Staubli VAL3: EnterPageKey.pgx

program EnterPageKey(num& x_nKey, num& x_nSelect, string& x_sItem)
  local string l_sStr
  local num l_nKey
  local string l_sEmpty
  local string l_sValue
  local num l_nItem
  local num l_nView
  local string l_sItem
  local point lp
  local string l_sYN[2]
  local bool l_bRes
begin
  //
  switch x_nSelect
    case 0
      if x_nKey==270
        call user:editNum(x_sItem,sListItemValue[x_nSelect],fFrame[sItem].trsf.x,x_nSelect)
      endIf
    break
    case 1
      if x_nKey==270
        call user:editNum(x_sItem,sListItemValue[x_nSelect],fFrame[sItem].trsf.y,x_nSelect)
      endIf
    break
    case 2
      if x_nKey==270
         call user:editNum(x_sItem,sListItemValue[x_nSelect],fFrame[sItem].trsf.z,x_nSelect)
      endIf
    break
    case 3
      if x_nKey==270
        call user:editNum(x_sItem,sListItemValue[x_nSelect],fFrame[sItem].trsf.rx,x_nSelect)
      endIf
    break
    case 4
      if x_nKey==27
         call user:editNum(x_sItem,sListItemValue[x_nSelect],fFrame[sItem].trsf.ry,x_nSelect)
      endIf
    break
    case 5
      if x_nKey==270
        call user:editNum(x_sItem,sListItemValue[x_nSelect],fFrame[sItem].trsf.rz,x_nSelect)
      endIf
    break
  endSwitch
  if x_nKey==270
    bUserRefresh=true
    bListRefresh=true
  endIf
end
